(* Schneider Machine Expert - Basic project State2_DrvObject_ModbusRTU, file version 2.7.0.0 *)
(* ProjectInformations: Name=New project *)

HARDWARE
  Cpu 0: TM221ME16T/G
  ModuleExtensionObject 0: TM3AM6/G
  EthernetConfiguration: NetworkName=M221, IpAllocationMode=FixedAddress, IpAddress=192.168.3.84, SubnetMask=255.255.255.0
  SerialLineConfiguration: Baud=Baud38400, Parity=ParityEven, DataBits=DataBits8, StopBits=StopBits1, PhysicalMedium=PhysicalMediumRs485, TransmissionMode=TransmissionModeIoScannerRtu
  MastTask: UsePeriodScanMode=true, PeriodScan=1
  FastTask: Period=255
  CpuBehavior: StartingMode=StartAsPreviousState, AutoSaveRamOnEeprom=true, WatchdogPeriod=250

SYMBOLS  (address, symbol, comment, settings)
  %M0       RUNMODE
  %M1       SW_FWD
  %M2       SW_BWD
  %M3       SW_RESET
  %M4       SW_POWER
  %M10      SL1_STATUS_STOPPED
  %M11      SL1_STATUS_INITREQED
  %M12      SL1_STATUS_OP
  %M13      SL1_STATUS_PARTIALLY_OP
  %M14      SL1_STATUS_SUSPENED
  %M15      ERRORRESET
  %M100     IO1_STATUS_VALID  "VALID"
  %M101     IO1_STATUS_ERRORSTOP  "ERRORSTOP"
  %M102     IO1_STATUS_DISABLED  "DISABLED"
  %M103     IO1_STATUS_STOPPING  "STOPPING"
  %M104     IO1_STATUS_STANDSTILL  "STANDSTILL"
  %M105     IO1_STATUS_CONTMOTION  "CONTMOTION"
  %M106     IO1_STATUS_ERROR  "ERROR"
  %M107     IO1_MC_RESET_DONE  "DONE"
  %M108     IO1_MC_RESET_BUSY  "BUSY"
  %M109     IO1_MC_RESET_ERROR  "ERROR"
  %M110     IO1_MC_POWER_STATUS
  %M111     IO1_MC_POWER_ERROR
  %M112     IO1_MC_JOG_DONE
  %M113     IO1_MC_JOG_BUSY
  %M114     IO1_MC_JOG_CMDABORTED
  %M115     IO1_MC_JOG_ERROR
  %M116     IO1_DRIVE_READY
  %M117     IO1_DRIVE_POWERON
  %M118     IO1_DRIVE_POWER_IL
  %M119     IO1_OP_IL
  %M120     IO1_JOG_FW
  %M121     IO1_JOG_BW
  %M122     IO1_MCREADMOTIONSTS_VALID
  %M123     IO1_MCREADMOTIONSTS_CONSTANTVEL
  %M124     IO1_MCREADMOTIONSTS_ACCELERATING
  %M125     IO1_MCREADMOTIONSTS_DECELERATING
  %M126     IO1_MCREADMOTIONSTS_ERROR
  %M127     IO1_MC_MOVEVEL_IL
  %M128     IO1_MC_MOVEVEL_CMD
  %M129     IO1_MC_MOVEVEL_CONTUPDATE
  %M130     IO1_MC_MOVEVEL_INVEL
  %M131     IO1_MC_MOVEVEL_BUSY
  %M132     IO1_MC_MOVEVEL_CMDABORTED
  %M133     IO1_MC_MOVEVEL_ERROR
  %M134     IO1_MC_STOP_IL
  %M135     IO1_MC_STOP_CMD
  %M136     IO1_MC_STOP_DONE
  %M137     IO1_MC_STOP_BUSY
  %M138     IO1_MC_STOP_ERROR
  %M139     IO1_POWER_RESET
  %S6       SB_TB1S  "Time base of 1 s generated by an internal clock"
  %S12      SB_RUNMODE  "The controller is running"
  %S107     SB_IOBUSRESTART  "The rising edge on this bit allows to reconfigure and restart the IO bus"
  %S110     SB_IOSCAN1RESET  "Set to 1 to reset the IOScanner on Serial Line 1"
  %SW210    SW_IOSCAN1STATUS  "Contains the IOScanner status of Serial Line 1"
  %MW0      MW_SLOT1_AO_CH0_SP
  %MW100    IO1_MC_POWER_ERRORID
  %MW101    IO1_MC_READSTATUS_ERRORID
  %MW102    IO1_MC_RESET_ERRORID
  %MW103    IO1_MC_JOG_ERRORID
  %MW104    IO1_MC_MOVEVEL_ERRORID
  %MW105    IO1_MC_STOP_ERRORID
  %MW106    IO1_ACTUALVEL
  %MW107    IO1_MC_READMOTIONSTATE_ERRORID
  %MW110    IO1_JOG_VEL
  %MW111    IO1_MOVEVEL_VEL
  %MF0      FLOAT_SETPOINT0
  %MC_JOG_ATV0 IO1_ATV320_MC_JOG  [Axis(Value(DriveAxis=DRV0)), Vel(Value(short=0))]
  %MC_MOVEVEL_ATV0 IO1_ATV320_MOVEVEL  [Axis(Value(DriveAxis=DRV0)), Vel(Value(short=0))]
  %MC_POWER_ATV0 IO1_MC_POWER  [Axis(Value(DriveAxis=DRV0))]
  %MC_READMOTIONSTATE_ATV0 IO1_ATV320_MC_READMOTIONSTATE  [Axis(Value(DriveAxis=DRV0))]
  %MC_READSTATUS_ATV0 IO1_ATV320_MC_READSTATUS  [Axis(Value(DriveAxis=DRV0))]
  %MC_RESET_ATV0 ATV320_1_MC_RESET  [Axis(Value(DriveAxis=DRV0))]
  %MC_STOP_ATV0 IO1_ATV320_MC_STOP  [Axis(Value(DriveAxis=DRV0))]
  %FB_SLSTATUS0 SL1_STATUS  [UserDefineFunctionPouName=FB_SLSTATUS]
  %I0.0     I_CH0_SW_FWD
  %I0.1     I_CH1_SW_BWD
  %I0.2     I_CH2_SW_RESET
  %I0.3     I_CH3_SW_POWERON
  %Q0.0     O_CH0_JOG_FW_CMD
  %Q0.1     O_CH1_JOG_BW_CMD
  %Q0.3     O_CH3_POWER_STATUS
  %IW1.0    SLOT1_AI_CHANNEL0  [Type=Type_0_10V, Scope=Scope_Customized, Minimum=0, Maximum=10000]
  %IW1.1    SLOT1_AI_CHANNEL1  [Type=Type_0_10V, Scope=Scope_Customized, Minimum=0, Maximum=10000]
  %IW1.2    SLOT1_AI_CHANNEL2  [Type=Type_0_10V, Scope=Scope_Customized, Minimum=0, Maximum=10000]
  %IW1.3    SLOT1_AI_CHANNEL3  [Type=Type_0_10V, Scope=Scope_Customized, Minimum=0, Maximum=10000]
  %QW1.0    SLOT1_AO_CHANNEL0  [Type=Type_0_10V, Scope=Scope_Customized, Minimum=0, Maximum=10000]
  %QW1.1    SLOT1_AO_CHANNEL1  [Type=Type_0_10V, Scope=Scope_Customized, Minimum=0, Maximum=10000]
  %DRV0     IO1_ATV320

POU Pou01_System
  (* SectionNumber=1 *)

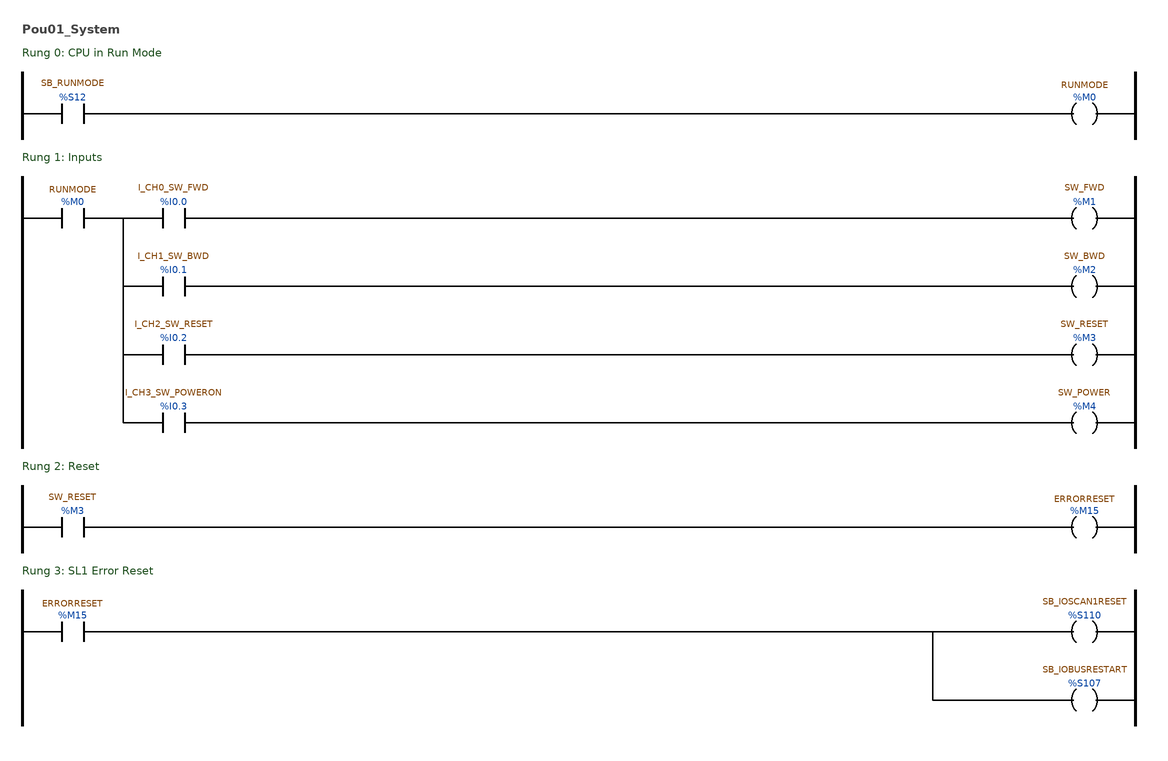

// Rung 0: CPU in Run Mode
  LD %S12                 (* SB_RUNMODE *)
  ST %M0                  (* RUNMODE *)
  // as ST:
  //   RUNMODE := SB_RUNMODE;

// Rung 1: Inputs
  LD %M0                  (* RUNMODE *)
  MPS
  AND %I0.0               (* I_CH0_SW_FWD *)
  ST %M1                  (* SW_FWD *)
  MRD
  AND %I0.1               (* I_CH1_SW_BWD *)
  ST %M2                  (* SW_BWD *)
  MRD
  AND %I0.2               (* I_CH2_SW_RESET *)
  ST %M3                  (* SW_RESET *)
  MPP
  AND %I0.3               (* I_CH3_SW_POWERON *)
  ST %M4                  (* SW_POWER *)
  // as ST:
  //   SW_FWD := RUNMODE AND I_CH0_SW_FWD;
  //   SW_BWD := RUNMODE AND I_CH1_SW_BWD;
  //   SW_RESET := RUNMODE AND I_CH2_SW_RESET;
  //   SW_POWER := RUNMODE AND I_CH3_SW_POWERON;

// Rung 2: Reset
  LD %M3                  (* SW_RESET *)
  ST %M15                 (* ERRORRESET *)
  // as ST:
  //   ERRORRESET := SW_RESET;

// Rung 3: SL1 Error Reset
  LD %M15                 (* ERRORRESET *)
  ST %S110                (* SB_IOSCAN1RESET *)
  ST %S107                (* SB_IOBUSRESTART *)
  // as ST:
  //   SB_IOSCAN1RESET := ERRORRESET;
  //   SB_IOBUSRESTART := ERRORRESET;

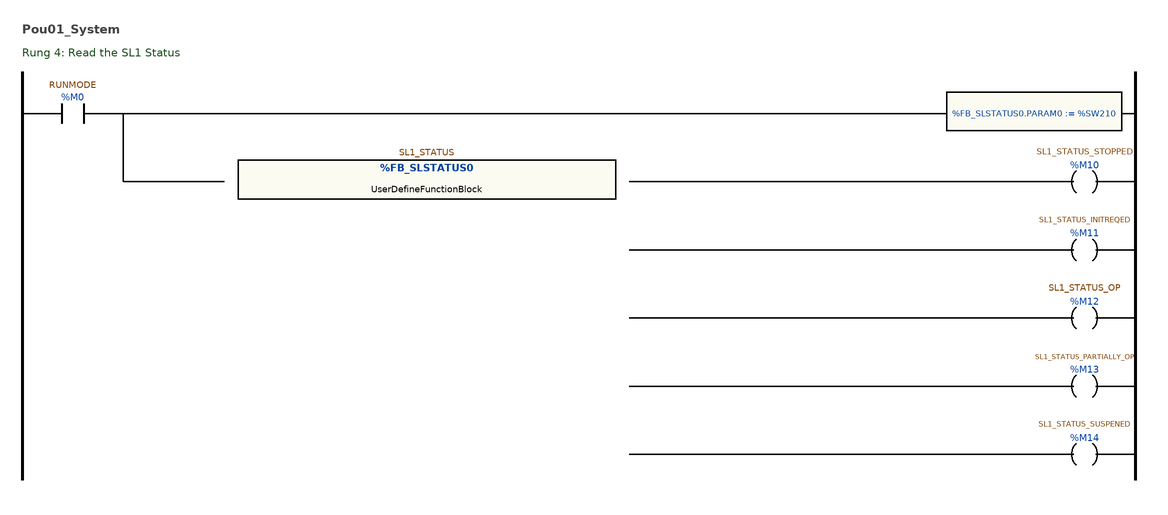

// Rung 4: Read the SL1 Status
  LD 1
  MULTIFB
  LD 1
  AND %M0                 (* RUNMODE *)
  ST %MW2009:X0
  LD %MW2009:X0
  [ %FB_SLSTATUS0.PARAM0 := %SW210 ](* SW_IOSCAN1STATUS *)
  BLK_UDFB 3
  LD %MW2009:X0
  ST %UDF1.PARAMW1:X0
  LD 1
  ST %UDF1.PARAMW1:X8
  [ %UDF1.PARAMW0 := %FB_SLSTATUS0.PARAM0 ]
  [ %UDF1.RETW0 := %UDF2.RETW0 ]
  [ %UDF1.RETW1 := %UDF2.RETW1 ]
  [ %UDF1.RETW2 := %UDF2.RETW2 ]
  [ %UDF1.RETW3 := %UDF2.RETW3 ]
  UDF1
  [ %UDF2.RETW0 := %UDF1.RETW0 ]
  [ %UDF2.RETW1 := %UDF1.RETW1 ]
  [ %UDF2.RETW2 := %UDF1.RETW2 ]
  [ %UDF2.RETW3 := %UDF1.RETW3 ]
  [ %FB_SLSTATUS0.PARAM0 := %UDF1.PARAMW0 ]
  LD %UDF1.RETW0:X0
  ST %M10                 (* SL1_STATUS_STOPPED *)
  LD %UDF1.RETW0:X1
  ST %M11                 (* SL1_STATUS_INITREQED *)
  LD %UDF1.RETW0:X2
  ST %M12                 (* SL1_STATUS_OP *)
  LD %UDF1.RETW0:X3
  ST %M13                 (* SL1_STATUS_PARTIALLY_OP *)
  LD %UDF1.RETW0:X4
  ST %M14                 (* SL1_STATUS_SUSPENED *)
  END_BLK_UDFB 3
  MULTIFB

POU Pou02_ATV320_1
  (* SectionNumber=2 *)

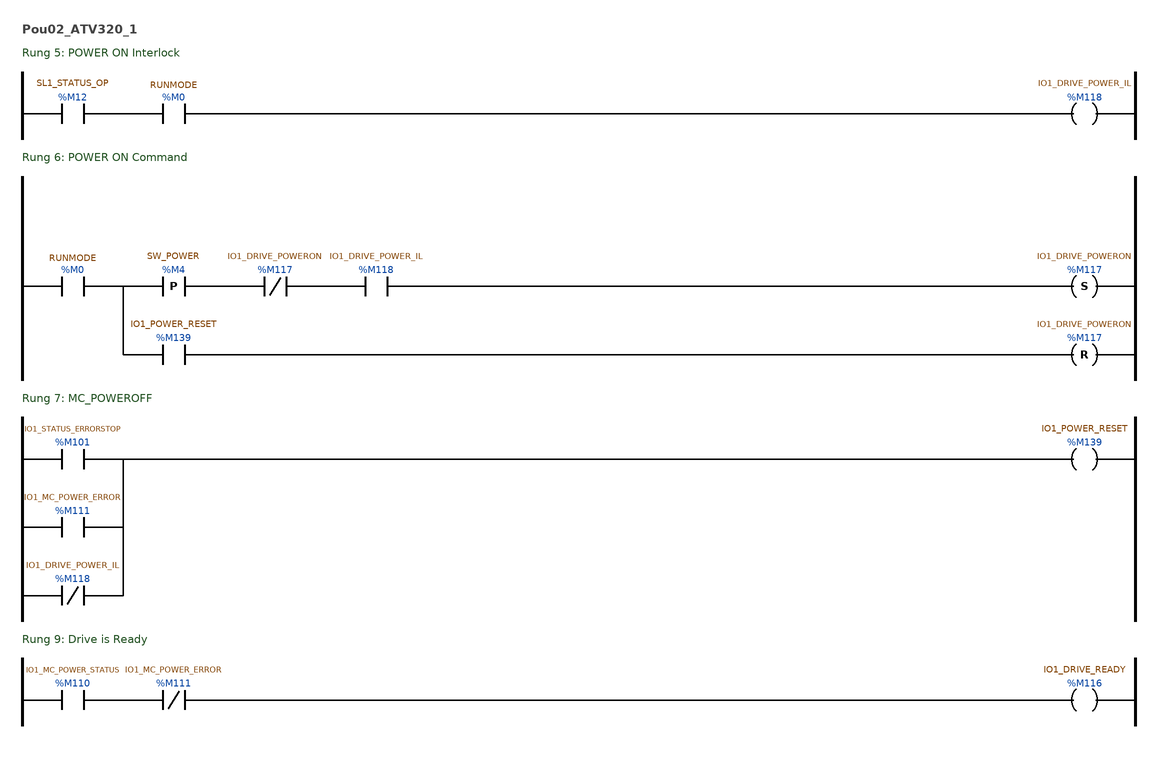

// Rung 5: POWER ON Interlock
  LD %M12                 (* SL1_STATUS_OP *)
  AND %M0                 (* RUNMODE *)
  ST %M118                (* IO1_DRIVE_POWER_IL *)
  // as ST:
  //   IO1_DRIVE_POWER_IL := SL1_STATUS_OP AND RUNMODE;

// Rung 6: POWER ON Command
  LD %M0                  (* RUNMODE *)
  MPS
  ANDR %M4                (* SW_POWER *)
  ANDN %M117              (* IO1_DRIVE_POWERON *)
  AND %M118               (* IO1_DRIVE_POWER_IL *)
  S %M117                 (* IO1_DRIVE_POWERON *)
  MPP
  AND %M139               (* IO1_POWER_RESET *)
  R %M117                 (* IO1_DRIVE_POWERON *)
  // as ST:
  //   IF RUNMODE AND RISING(SW_POWER) AND NOT IO1_DRIVE_POWERON AND IO1_DRIVE_POWER_IL THEN IO1_DRIVE_POWERON := TRUE; END_IF;
  //   IF RUNMODE AND IO1_POWER_RESET THEN IO1_DRIVE_POWERON := FALSE; END_IF;

// Rung 7: MC_POWEROFF
  LD %M101                (* IO1_STATUS_ERRORSTOP *)
  OR %M111                (* IO1_MC_POWER_ERROR *)
  ORN %M118               (* IO1_DRIVE_POWER_IL *)
  ST %M139                (* IO1_POWER_RESET *)
  // as ST:
  //   IO1_POWER_RESET := IO1_STATUS_ERRORSTOP OR IO1_MC_POWER_ERROR OR NOT IO1_DRIVE_POWER_IL;

// Rung 8: MC_POWER
  LD 1
  MULTIFB
  LD 1
  AND %M117               (* IO1_DRIVE_POWERON *)
  ST %MW2009:X0
  BLK %MC_POWER_ATV0
  LD %MW2009:X0
  ENABLE
  OUT_BLK
  LD STATUS
  ST %M110                (* IO1_MC_POWER_STATUS *)
  LD ERROR
  ST %M111                (* IO1_MC_POWER_ERROR *)
  END_BLK
  LD %MW2009:X0
  [ %MW100 := %MC_POWER_ATV0.ERRORID ](* IO1_MC_POWER_ERRORID *)
  MULTIFB
  // as ST:
  //   %MC_POWER_ATV0(ENABLE := IO1_DRIVE_POWERON);
  //   IO1_MC_POWER_STATUS := %MC_POWER_ATV0.STATUS;
  //   IO1_MC_POWER_ERROR := %MC_POWER_ATV0.ERROR;
  //   IF IO1_DRIVE_POWERON THEN IO1_MC_POWER_ERRORID := %MC_POWER_ATV0.ERRORID; END_IF;
  (* the ladder stored for this rung does not match its IL; not drawn *)

// Rung 9: Drive is Ready
  LD %M110                (* IO1_MC_POWER_STATUS *)
  ANDN %M111              (* IO1_MC_POWER_ERROR *)
  ST %M116                (* IO1_DRIVE_READY *)
  // as ST:
  //   IO1_DRIVE_READY := IO1_MC_POWER_STATUS AND NOT IO1_MC_POWER_ERROR;

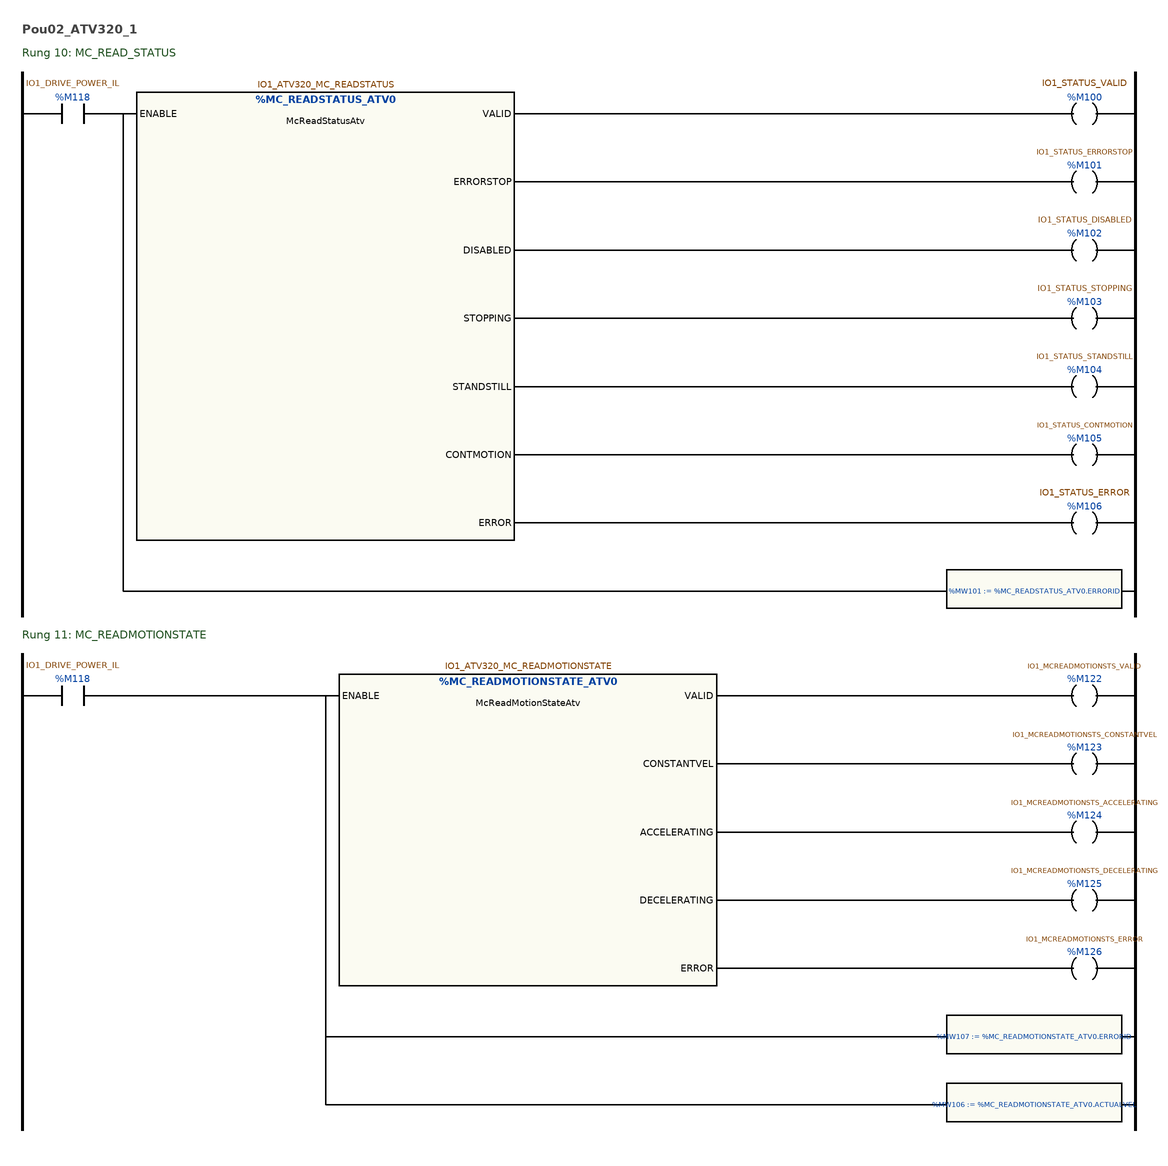

// Rung 10: MC_READ_STATUS
  LD 1
  MULTIFB
  LD 1
  AND %M118               (* IO1_DRIVE_POWER_IL *)
  ST %MW2009:X0
  BLK %MC_READSTATUS_ATV0
  LD %MW2009:X0
  ENABLE
  OUT_BLK
  LD VALID
  ST %M100                (* IO1_STATUS_VALID *)
  LD ERRORSTOP
  ST %M101                (* IO1_STATUS_ERRORSTOP *)
  LD DISABLED
  ST %M102                (* IO1_STATUS_DISABLED *)
  LD STOPPING
  ST %M103                (* IO1_STATUS_STOPPING *)
  LD STANDSTILL
  ST %M104                (* IO1_STATUS_STANDSTILL *)
  LD CONTMOTION
  ST %M105                (* IO1_STATUS_CONTMOTION *)
  LD ERROR
  ST %M106                (* IO1_STATUS_ERROR *)
  END_BLK
  LD %MW2009:X0
  [ %MW101 := %MC_READSTATUS_ATV0.ERRORID ](* IO1_MC_READSTATUS_ERRORID *)
  MULTIFB
  // as ST:
  //   %MC_READSTATUS_ATV0(ENABLE := IO1_DRIVE_POWER_IL);
  //   IO1_STATUS_VALID := %MC_READSTATUS_ATV0.VALID;
  //   IO1_STATUS_ERRORSTOP := %MC_READSTATUS_ATV0.ERRORSTOP;
  //   IO1_STATUS_DISABLED := %MC_READSTATUS_ATV0.DISABLED;
  //   IO1_STATUS_STOPPING := %MC_READSTATUS_ATV0.STOPPING;
  //   IO1_STATUS_STANDSTILL := %MC_READSTATUS_ATV0.STANDSTILL;
  //   IO1_STATUS_CONTMOTION := %MC_READSTATUS_ATV0.CONTMOTION;
  //   IO1_STATUS_ERROR := %MC_READSTATUS_ATV0.ERROR;
  //   IF IO1_DRIVE_POWER_IL THEN IO1_MC_READSTATUS_ERRORID := %MC_READSTATUS_ATV0.ERRORID; END_IF;

// Rung 11: MC_READMOTIONSTATE
  LD 1
  MULTIFB
  LD 1
  AND %M118               (* IO1_DRIVE_POWER_IL *)
  ST %MW2009:X0
  BLK %MC_READMOTIONSTATE_ATV0
  LD %MW2009:X0
  ENABLE
  OUT_BLK
  LD VALID
  ST %M122                (* IO1_MCREADMOTIONSTS_VALID *)
  LD CONSTANTVEL
  ST %M123                (* IO1_MCREADMOTIONSTS_CONSTANTVEL *)
  LD ACCELERATING
  ST %M124                (* IO1_MCREADMOTIONSTS_ACCELERATING *)
  LD DECELERATING
  ST %M125                (* IO1_MCREADMOTIONSTS_DECELERATING *)
  LD ERROR
  ST %M126                (* IO1_MCREADMOTIONSTS_ERROR *)
  END_BLK
  LD %MW2009:X0
  [ %MW107 := %MC_READMOTIONSTATE_ATV0.ERRORID ](* IO1_MC_READMOTIONSTATE_ERRORID *)
  [ %MW106 := %MC_READMOTIONSTATE_ATV0.ACTUALVEL ](* IO1_ACTUALVEL *)
  MULTIFB
  // as ST:
  //   %MC_READMOTIONSTATE_ATV0(ENABLE := IO1_DRIVE_POWER_IL);
  //   IO1_MCREADMOTIONSTS_VALID := %MC_READMOTIONSTATE_ATV0.VALID;
  //   IO1_MCREADMOTIONSTS_CONSTANTVEL := %MC_READMOTIONSTATE_ATV0.CONSTANTVEL;
  //   IO1_MCREADMOTIONSTS_ACCELERATING := %MC_READMOTIONSTATE_ATV0.ACCELERATING;
  //   IO1_MCREADMOTIONSTS_DECELERATING := %MC_READMOTIONSTATE_ATV0.DECELERATING;
  //   IO1_MCREADMOTIONSTS_ERROR := %MC_READMOTIONSTATE_ATV0.ERROR;
  //   IF IO1_DRIVE_POWER_IL THEN IO1_MC_READMOTIONSTATE_ERRORID := %MC_READMOTIONSTATE_ATV0.ERRORID; END_IF;
  //   IF IO1_DRIVE_POWER_IL THEN IO1_ACTUALVEL := %MC_READMOTIONSTATE_ATV0.ACTUALVEL; END_IF;

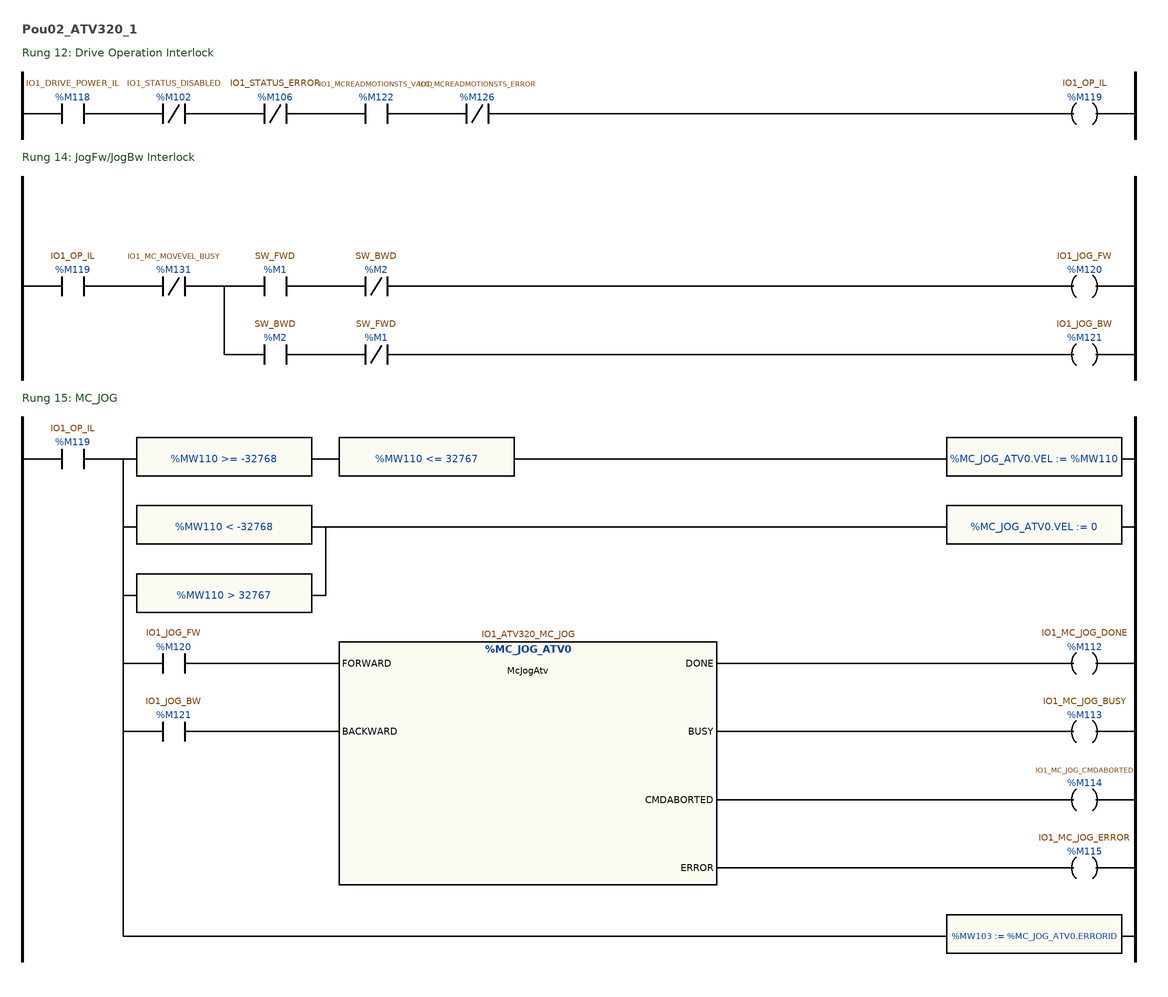

// Rung 12: Drive Operation Interlock
  LD %M118                (* IO1_DRIVE_POWER_IL *)
  ANDN %M102              (* IO1_STATUS_DISABLED *)
  ANDN %M106              (* IO1_STATUS_ERROR *)
  AND %M122               (* IO1_MCREADMOTIONSTS_VALID *)
  ANDN %M126              (* IO1_MCREADMOTIONSTS_ERROR *)
  ST %M119                (* IO1_OP_IL *)
  // as ST:
  //   IO1_OP_IL := IO1_DRIVE_POWER_IL AND NOT IO1_STATUS_DISABLED AND NOT IO1_STATUS_ERROR AND IO1_MCREADMOTIONSTS_VALID AND NOT IO1_MCREADMOTIONSTS_ERROR;

// Rung 13: MC_RESET
  LD 1
  MULTIFB
  LD 1
  AND %M0                 (* RUNMODE *)
  AND %M15                (* ERRORRESET *)
  ST %MW2009:X0
  BLK %MC_RESET_ATV0
  LD %MW2009:X0
  EXECUTE
  OUT_BLK
  LD DONE
  ST %M107                (* IO1_MC_RESET_DONE *)
  LD BUSY
  ST %M108                (* IO1_MC_RESET_BUSY *)
  LD ERROR
  ST %M109                (* IO1_MC_RESET_ERROR *)
  END_BLK
  LD %MW2009:X0
  [ %MW102 := %MC_RESET_ATV0.ERRORID ](* IO1_MC_RESET_ERRORID *)
  MULTIFB
  // as ST:
  //   %MC_RESET_ATV0(EXECUTE := RUNMODE AND ERRORRESET);
  //   IO1_MC_RESET_DONE := %MC_RESET_ATV0.DONE;
  //   IO1_MC_RESET_BUSY := %MC_RESET_ATV0.BUSY;
  //   IO1_MC_RESET_ERROR := %MC_RESET_ATV0.ERROR;
  //   IF RUNMODE AND ERRORRESET THEN IO1_MC_RESET_ERRORID := %MC_RESET_ATV0.ERRORID; END_IF;
  (* the ladder stored for this rung does not match its IL; not drawn *)

// Rung 14: JogFw/JogBw Interlock
  LD %M119                (* IO1_OP_IL *)
  ANDN %M131              (* IO1_MC_MOVEVEL_BUSY *)
  MPS
  AND %M1                 (* SW_FWD *)
  ANDN %M2                (* SW_BWD *)
  ST %M120                (* IO1_JOG_FW *)
  MPP
  AND %M2                 (* SW_BWD *)
  ANDN %M1                (* SW_FWD *)
  ST %M121                (* IO1_JOG_BW *)
  // as ST:
  //   IO1_JOG_FW := IO1_OP_IL AND NOT IO1_MC_MOVEVEL_BUSY AND SW_FWD AND NOT SW_BWD;
  //   IO1_JOG_BW := IO1_OP_IL AND NOT IO1_MC_MOVEVEL_BUSY AND SW_BWD AND NOT SW_FWD;

// Rung 15: MC_JOG
  LD 1
  MULTIFB
  LD 1
  AND %M119               (* IO1_OP_IL *)
  ST %MW2009:X0
  LD %MW2009:X0
  MPS
  AND [ %MW110 >= -32768 ](* IO1_JOG_VEL *)
  AND [ %MW110 <= 32767 ] (* IO1_JOG_VEL *)
  [ %MC_JOG_ATV0.VEL := %MW110 ](* IO1_JOG_VEL *)
  MPP
  AND( [ %MW110 < -32768 ](* IO1_JOG_VEL *)
  OR [ %MW110 > 32767 ]   (* IO1_JOG_VEL *)
  )
  [ %MC_JOG_ATV0.VEL := 0 ]
  BLK %MC_JOG_ATV0
  LD %MW2009:X0
  MPS
  AND %M120               (* IO1_JOG_FW *)
  FORWARD
  MPP
  AND %M121               (* IO1_JOG_BW *)
  BACKWARD
  OUT_BLK
  LD DONE
  ST %M112                (* IO1_MC_JOG_DONE *)
  LD BUSY
  ST %M113                (* IO1_MC_JOG_BUSY *)
  LD CMDABORTED
  ST %M114                (* IO1_MC_JOG_CMDABORTED *)
  LD ERROR
  ST %M115                (* IO1_MC_JOG_ERROR *)
  END_BLK
  LD %MW2009:X0
  [ %MW103 := %MC_JOG_ATV0.ERRORID ](* IO1_MC_JOG_ERRORID *)
  MULTIFB
  // as ST:
  //   IF IO1_OP_IL AND IO1_JOG_VEL >= -32768 AND IO1_JOG_VEL <= 32767 THEN %MC_JOG_ATV0.VEL := IO1_JOG_VEL; END_IF;
  //   IF IO1_OP_IL AND (IO1_JOG_VEL < -32768 OR IO1_JOG_VEL > 32767) THEN %MC_JOG_ATV0.VEL := 0; END_IF;
  //   %MC_JOG_ATV0(FORWARD := IO1_OP_IL AND IO1_JOG_FW, BACKWARD := IO1_OP_IL AND IO1_JOG_BW);
  //   IO1_MC_JOG_DONE := %MC_JOG_ATV0.DONE;
  //   IO1_MC_JOG_BUSY := %MC_JOG_ATV0.BUSY;
  //   IO1_MC_JOG_CMDABORTED := %MC_JOG_ATV0.CMDABORTED;
  //   IO1_MC_JOG_ERROR := %MC_JOG_ATV0.ERROR;
  //   IF IO1_OP_IL THEN IO1_MC_JOG_ERRORID := %MC_JOG_ATV0.ERRORID; END_IF;

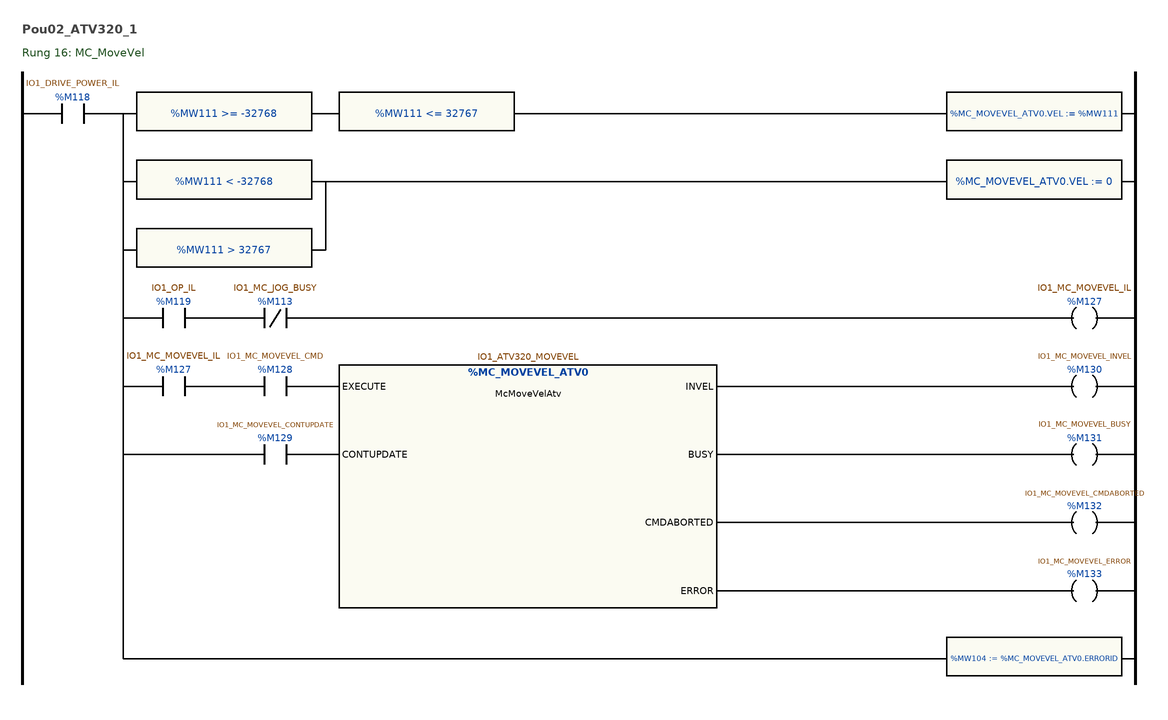

// Rung 16: MC_MoveVel
  LD 1
  MULTIFB
  LD 1
  AND %M118               (* IO1_DRIVE_POWER_IL *)
  ST %MW2009:X0
  LD %MW2009:X0
  MPS
  AND [ %MW111 >= -32768 ](* IO1_MOVEVEL_VEL *)
  AND [ %MW111 <= 32767 ] (* IO1_MOVEVEL_VEL *)
  [ %MC_MOVEVEL_ATV0.VEL := %MW111 ](* IO1_MOVEVEL_VEL *)
  MRD
  AND( [ %MW111 < -32768 ](* IO1_MOVEVEL_VEL *)
  OR [ %MW111 > 32767 ]   (* IO1_MOVEVEL_VEL *)
  )
  [ %MC_MOVEVEL_ATV0.VEL := 0 ]
  MPP
  AND %M119               (* IO1_OP_IL *)
  ANDN %M113              (* IO1_MC_JOG_BUSY *)
  ST %M127                (* IO1_MC_MOVEVEL_IL *)
  BLK %MC_MOVEVEL_ATV0
  LD %MW2009:X0
  MPS
  AND %M127               (* IO1_MC_MOVEVEL_IL *)
  AND %M128               (* IO1_MC_MOVEVEL_CMD *)
  EXECUTE
  MPP
  AND %M129               (* IO1_MC_MOVEVEL_CONTUPDATE *)
  CONTUPDATE
  OUT_BLK
  LD INVEL
  ST %M130                (* IO1_MC_MOVEVEL_INVEL *)
  LD BUSY
  ST %M131                (* IO1_MC_MOVEVEL_BUSY *)
  LD CMDABORTED
  ST %M132                (* IO1_MC_MOVEVEL_CMDABORTED *)
  LD ERROR
  ST %M133                (* IO1_MC_MOVEVEL_ERROR *)
  END_BLK
  LD %MW2009:X0
  [ %MW104 := %MC_MOVEVEL_ATV0.ERRORID ](* IO1_MC_MOVEVEL_ERRORID *)
  MULTIFB
  // as ST:
  //   IF IO1_DRIVE_POWER_IL AND IO1_MOVEVEL_VEL >= -32768 AND IO1_MOVEVEL_VEL <= 32767 THEN %MC_MOVEVEL_ATV0.VEL := IO1_MOVEVEL_VEL; END_IF;
  //   IF IO1_DRIVE_POWER_IL AND (IO1_MOVEVEL_VEL < -32768 OR IO1_MOVEVEL_VEL > 32767) THEN %MC_MOVEVEL_ATV0.VEL := 0; END_IF;
  //   IO1_MC_MOVEVEL_IL := IO1_DRIVE_POWER_IL AND IO1_OP_IL AND NOT IO1_MC_JOG_BUSY;
  //   %MC_MOVEVEL_ATV0(EXECUTE := IO1_DRIVE_POWER_IL AND IO1_MC_MOVEVEL_IL AND IO1_MC_MOVEVEL_CMD, CONTUPDATE := IO1_DRIVE_POWER_IL AND IO1_MC_MOVEVEL_CONTUPDATE);
  //   IO1_MC_MOVEVEL_INVEL := %MC_MOVEVEL_ATV0.INVEL;
  //   IO1_MC_MOVEVEL_BUSY := %MC_MOVEVEL_ATV0.BUSY;
  //   IO1_MC_MOVEVEL_CMDABORTED := %MC_MOVEVEL_ATV0.CMDABORTED;
  //   IO1_MC_MOVEVEL_ERROR := %MC_MOVEVEL_ATV0.ERROR;
  //   IF IO1_DRIVE_POWER_IL THEN IO1_MC_MOVEVEL_ERRORID := %MC_MOVEVEL_ATV0.ERRORID; END_IF;

// Rung 17: MC_STOP
  LD 1
  MULTIFB
  LD 1
  AND %M118               (* IO1_DRIVE_POWER_IL *)
  ST %MW2009:X0
  LD %MW2009:X0
  ST %M134                (* IO1_MC_STOP_IL *)
  BLK %MC_STOP_ATV0
  LD %MW2009:X0
  AND %M134               (* IO1_MC_STOP_IL *)
  AND %M135               (* IO1_MC_STOP_CMD *)
  EXECUTE
  OUT_BLK
  LD DONE
  ST %M136                (* IO1_MC_STOP_DONE *)
  LD BUSY
  ST %M137                (* IO1_MC_STOP_BUSY *)
  LD ERROR
  ST %M138                (* IO1_MC_STOP_ERROR *)
  END_BLK
  LD %MW2009:X0
  [ %MW105 := %MC_STOP_ATV0.ERRORID ](* IO1_MC_STOP_ERRORID *)
  MULTIFB
  // as ST:
  //   IO1_MC_STOP_IL := IO1_DRIVE_POWER_IL;
  //   %MC_STOP_ATV0(EXECUTE := IO1_DRIVE_POWER_IL AND IO1_MC_STOP_IL AND IO1_MC_STOP_CMD);
  //   IO1_MC_STOP_DONE := %MC_STOP_ATV0.DONE;
  //   IO1_MC_STOP_BUSY := %MC_STOP_ATV0.BUSY;
  //   IO1_MC_STOP_ERROR := %MC_STOP_ATV0.ERROR;
  //   IF IO1_DRIVE_POWER_IL THEN IO1_MC_STOP_ERRORID := %MC_STOP_ATV0.ERRORID; END_IF;
  (* the ladder stored for this rung does not match its IL; not drawn *)

POU Pou03_Outputs
  (* SectionNumber=3 *)

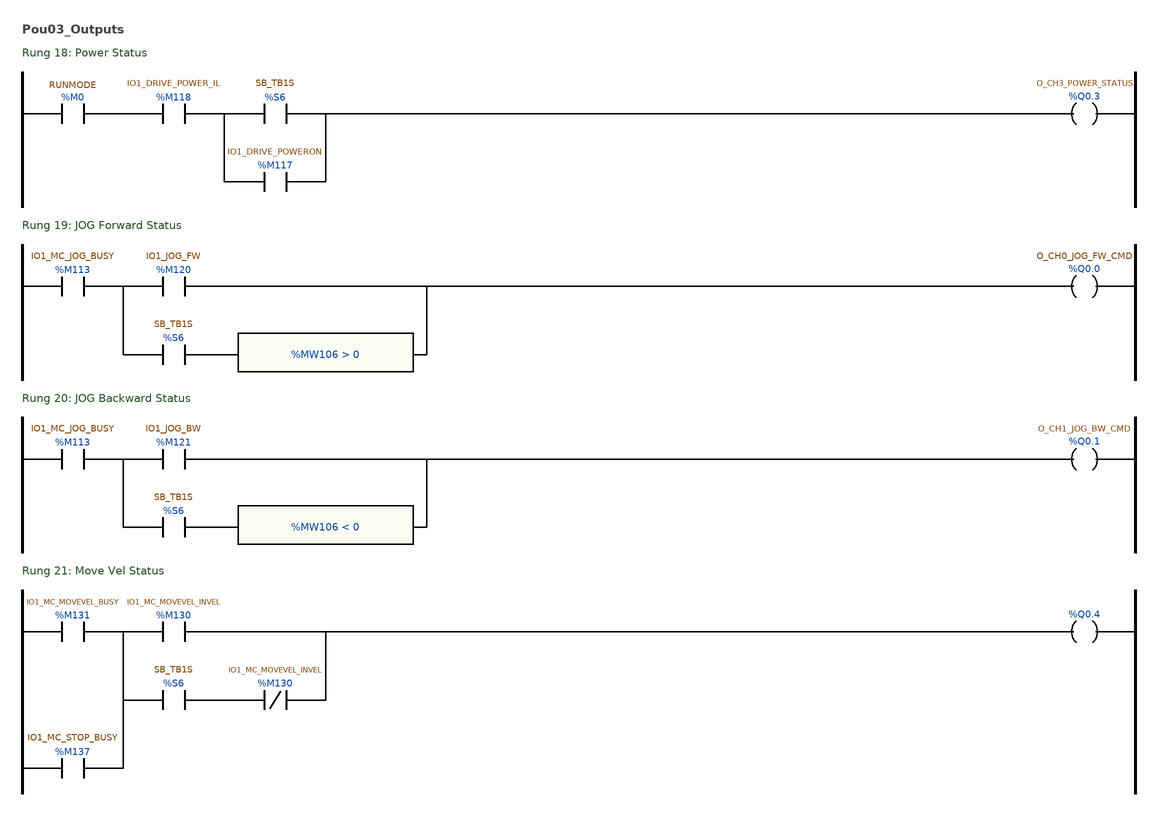

// Rung 18: Power Status
  LD %M0                  (* RUNMODE *)
  AND %M118               (* IO1_DRIVE_POWER_IL *)
  AND( %S6                (* SB_TB1S *)
  OR %M117                (* IO1_DRIVE_POWERON *)
  )
  ST %Q0.3                (* O_CH3_POWER_STATUS *)
  // as ST:
  //   O_CH3_POWER_STATUS := RUNMODE AND IO1_DRIVE_POWER_IL AND (SB_TB1S OR IO1_DRIVE_POWERON);

// Rung 19: JOG Forward Status
  LD %M113                (* IO1_MC_JOG_BUSY *)
  AND( %M120              (* IO1_JOG_FW *)
  OR( %S6                 (* SB_TB1S *)
  AND [ %MW106 > 0 ]      (* IO1_ACTUALVEL *)
  )
  )
  ST %Q0.0                (* O_CH0_JOG_FW_CMD *)
  // as ST:
  //   O_CH0_JOG_FW_CMD := IO1_MC_JOG_BUSY AND (IO1_JOG_FW OR SB_TB1S AND IO1_ACTUALVEL > 0);

// Rung 20: JOG Backward Status
  LD %M113                (* IO1_MC_JOG_BUSY *)
  AND( %M121              (* IO1_JOG_BW *)
  OR( %S6                 (* SB_TB1S *)
  AND [ %MW106 < 0 ]      (* IO1_ACTUALVEL *)
  )
  )
  ST %Q0.1                (* O_CH1_JOG_BW_CMD *)
  // as ST:
  //   O_CH1_JOG_BW_CMD := IO1_MC_JOG_BUSY AND (IO1_JOG_BW OR SB_TB1S AND IO1_ACTUALVEL < 0);

// Rung 21: Move Vel Status
  LD %M131                (* IO1_MC_MOVEVEL_BUSY *)
  OR %M137                (* IO1_MC_STOP_BUSY *)
  AND( %M130              (* IO1_MC_MOVEVEL_INVEL *)
  OR( %S6                 (* SB_TB1S *)
  ANDN %M130              (* IO1_MC_MOVEVEL_INVEL *)
  )
  )
  ST %Q0.4
  // as ST:
  //   %Q0.4 := (IO1_MC_MOVEVEL_BUSY OR IO1_MC_STOP_BUSY) AND (IO1_MC_MOVEVEL_INVEL OR SB_TB1S AND NOT IO1_MC_MOVEVEL_INVEL);

UserFunctionPou FC_SCALING2AO
  (* SectionNumber=4 *)

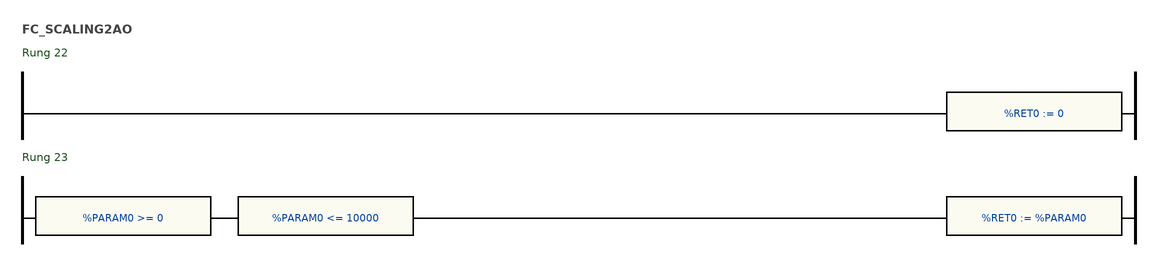

// Rung 22
  LD 1
  [ %RET0 := 0 ]
  // as ST:
  //   %RET0 := 0;

// Rung 23
  LD [ %PARAM0 >= 0 ]
  AND [ %PARAM0 <= 10000 ]
  [ %RET0 := %PARAM0 ]
  // as ST:
  //   IF %PARAM0 >= 0 AND %PARAM0 <= 10000 THEN %RET0 := %PARAM0; END_IF;

UserFunctionBlockPou FB_SLSTATUS
  (* SectionNumber=5 *)

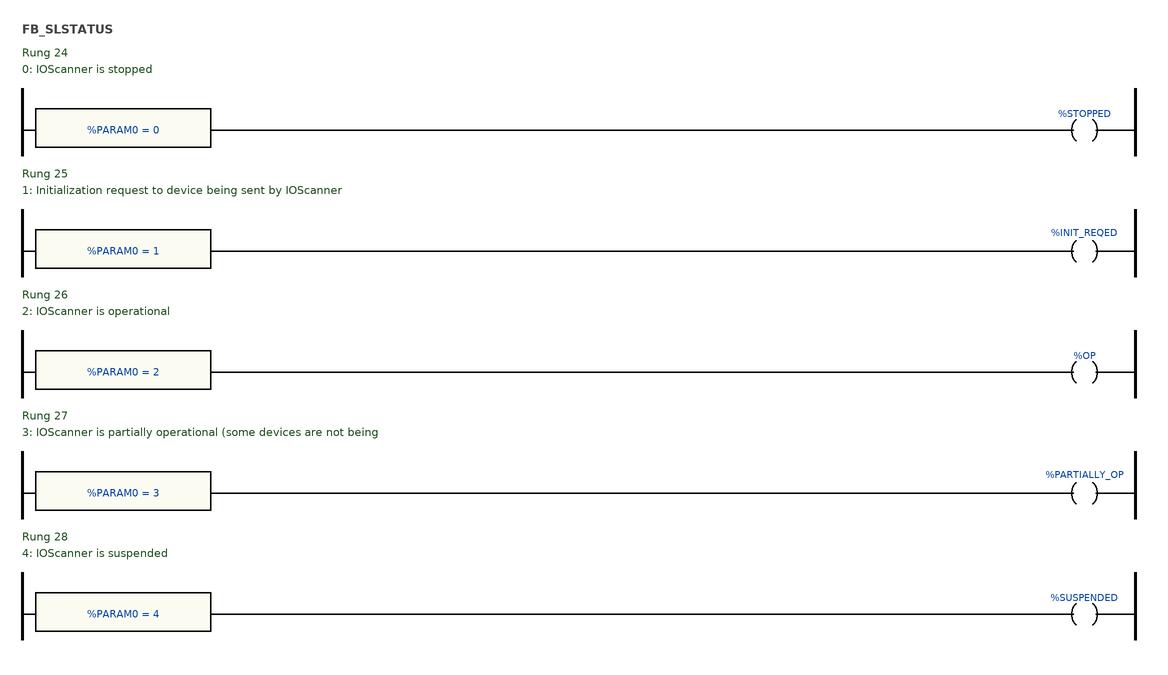

// Rung 24
// 0: IOScanner is stopped
  LD [ %PARAM0 = 0 ]
  ST %STOPPED
  // as ST:
  //   %STOPPED := %PARAM0 = 0;

// Rung 25
// 1: Initialization request to device being sent by IOScanner
  LD [ %PARAM0 = 1 ]
  ST %INIT_REQED
  // as ST:
  //   %INIT_REQED := %PARAM0 = 1;

// Rung 26
// 2: IOScanner is operational
  LD [ %PARAM0 = 2 ]
  ST %OP
  // as ST:
  //   %OP := %PARAM0 = 2;

// Rung 27
// 3: IOScanner is partially operational (some devices are not being
  LD [ %PARAM0 = 3 ]
  ST %PARTIALLY_OP
  // as ST:
  //   %PARTIALLY_OP := %PARAM0 = 3;

// Rung 28
// 4: IOScanner is suspended
  LD [ %PARAM0 = 4 ]
  ST %SUSPENDED
  // as ST:
  //   %SUSPENDED := %PARAM0 = 4;
